INTERFACE I_RepeatedField

METHOD CalculatePackedDataSize : HRESULT
VAR_OUTPUT
    nPackedDataSize : UDINT;
END_VAR
END_METHOD

METHOD CalculateSize : HRESULT

VAR_OUTPUT
	nSize : UDINT;
END_VAR
END_METHOD

METHOD ElementAtIndex : T_ANY
VAR_INPUT
	nIndex		: UDINT;
END_VAR
END_METHOD

PROPERTY ipFieldCodec : I_FieldCodec
GET
END_GET
END_PROPERTY

PROPERTY nCapcacity : UDINT
GET
END_GET
END_PROPERTY

PROPERTY nCount : UDINT
GET
END_GET
SET
END_SET
END_PROPERTY

METHOD SetValue : HRESULT
VAR_INPUT
	anyValue	: T_ANY;
END_VAR
END_METHOD

END_INTERFACE

(* stored: Version 1.1.0.1
   Itf I_RepeatedField: Id {df287fba-c0ab-4d65-bbd3-aa9b11c253c5}
   Method CalculatePackedDataSize: Id {e5b4cca5-e8f8-4023-8274-715fdfd4c456}
   Method CalculateSize: Id {7131302d-4e7f-40e9-ac93-ed1dc95621e5}
   Method ElementAtIndex: Id {811730db-b114-46ba-8b85-1b8fffa011d8}
   Property ipFieldCodec: Id {77aead32-80b0-4b85-a8ea-2e22373bbd25}
   Get Get: Id {f7aee202-98c4-4bf3-8440-204f034e065b}
   Property nCapcacity: Id {4914541c-9d02-48cf-8983-8f50db23c15b}
   Get Get: Id {e9413b38-69c2-4619-af78-34c77feb1c35}
   Property nCount: Id {a7e19284-ec89-4001-9bd9-258e5e66966e}
   Get Get: Id {6e0af163-7a85-41f2-a729-f468ec5e1d22}
   Set Set: Id {47979acb-e7c8-45ac-8257-73f8a8fcbaca}
   Method SetValue: Id {04df43e2-7f98-460e-a299-274520714bef} *)
